{attribute 'qualified_only'}
VAR_GLOBAL
	bAnalog_Inputs AT %I* : ARRAY[1..4] OF INT;
END_VAR

(* stored: Version 1.1.0.1, ProductVersion 3.1.4024.12
   GVL GVL: Id {844cf94b-bd0a-4a68-bff0-d37a51a5b111} *)
